FUNCTION_BLOCK FB_A IMPLEMENTS I_Name

VAR
    sVar1 : STRING := 'My name is A.';
END_VAR

{warning 'add property implementation'}
PROPERTY Name : STRING
GET
Name := sVar1;
END_GET
SET
sVar1 := Name;
END_SET
END_PROPERTY

END_FUNCTION_BLOCK

(* stored: Version 1.1.0.1, ProductVersion 3.1.4024.12
   POU FB_A: Id {35e748e4-3349-4454-ac4a-a44dffb5e8f1}, SpecialFunc None
   Property Name: Id {c6cafcbd-13e4-41c0-8209-8cb893a55895}
   Get Get: Id {f0aefa2c-f863-41ad-a042-591bef54ffe8}
   Set Set: Id {a8d9d6a7-e057-4e91-9e95-e9dea6813ed5} *)
